FUNCTION TryConvert_DWORD_TO_DWORD : BOOL
VAR_INPUT
	in : DWORD;
	out : REFERENCE TO DWORD;
END_VAR

out := in;
TryConvert_DWORD_TO_DWORD := TRUE;

END_FUNCTION

(* stored: Version 1.1.0.1, ProductVersion 3.1.4024.12
   POU TryConvert_DWORD_TO_DWORD: Id {8056e80c-d056-444b-a4e1-f8928a69dfa4}, SpecialFunc None *)
